SUBAPPLICATION Uebung_074 (* RPTO auf UT ausgeben mit Fendt-Schaltung *)
  (* Standard: 61499-2; Description: Copyright (c) 2023 Meisterschulen am Ostbahnhof This program and the accompanying materials are made available under the terms of the Eclipse Public License 2.0 which is available at https://www.eclipse.org/legal/epl-2.0/ SPDX-License-Identifier: EPL-2.0 *)
  (* Version 1.0, 2023-10-23, Franz Höpfinger, Meisterschulen am Ostbahnhof, initial API and implementation and/or initial documentation *)
  PACKAGE Uebungen;
  IMPORT Uebungen::const::UT::TECU::DefaultPool_TECU::NumberVariable_Rear_PTO_output_shaft_speed;
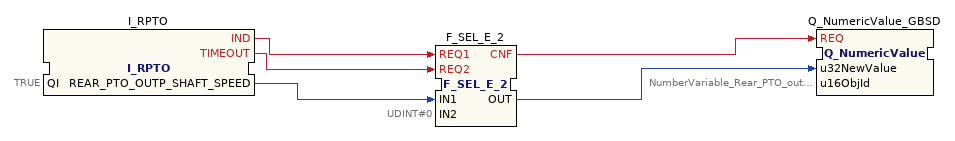
  (* "Fendt" Schaltung! *)
  FBS
    I_RPTO : isobus::tecu::I_RPTO(QI := TRUE);
    Q_NumericValue_GBSD : isobus::UT::Q::Q_NumericValue(u16ObjId := NumberVariable_Rear_PTO_output_shaft_speed);
    F_SEL_E_2 : eclipse4diac::utils::selection::F_SEL_E_2(IN2 := UDINT#0);
  END_FBS
  EVENT_CONNECTIONS
    I_RPTO.IND TO F_SEL_E_2.REQ1;
    F_SEL_E_2.CNF TO Q_NumericValue_GBSD.REQ;
    I_RPTO.TIMEOUT TO F_SEL_E_2.REQ2;
  END_CONNECTIONS
  DATA_CONNECTIONS
    I_RPTO.REAR_PTO_OUTP_SHAFT_SPEED TO F_SEL_E_2.IN1;
    F_SEL_E_2.OUT TO Q_NumericValue_GBSD.u32NewValue;
  END_CONNECTIONS
END_SUBAPPLICATION
